TYPE ST_AdsAddr :
STRUCT

	netId									:AMSNETID;
	port									:WORD;

END_STRUCT
END_TYPE

(* stored: Version 1.1.0.1, ProductVersion 3.1.4022.16
   DUT ST_AdsAddr: Id {c97e4cdf-7dcf-463c-9eca-9bad82d05ea0} *)
